FUNCTION_BLOCK Solenoid
VAR_INPUT

END_VAR
VAR_OUTPUT
END_VAR
VAR
END_VAR

END_FUNCTION_BLOCK

(* stored: Version 1.1.0.1, ProductVersion 3.1.4024.12
   POU Solenoid: Id {a1565ff4-83c0-4d25-afd3-9bce02147dc7}, SpecialFunc None *)
